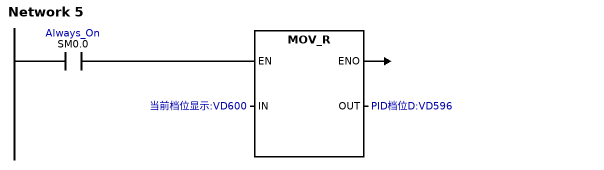
[picture p24: SBR12 networks 5-5]
Network 5
LD     Always_On:SM0.0
MOVR   当前档位显示:VD600, PID档位D:VD596
END_SUBROUTINE_BLOCK

SUBROUTINE_BLOCK PID换算档位:SBR13
TITLE=
BEGIN
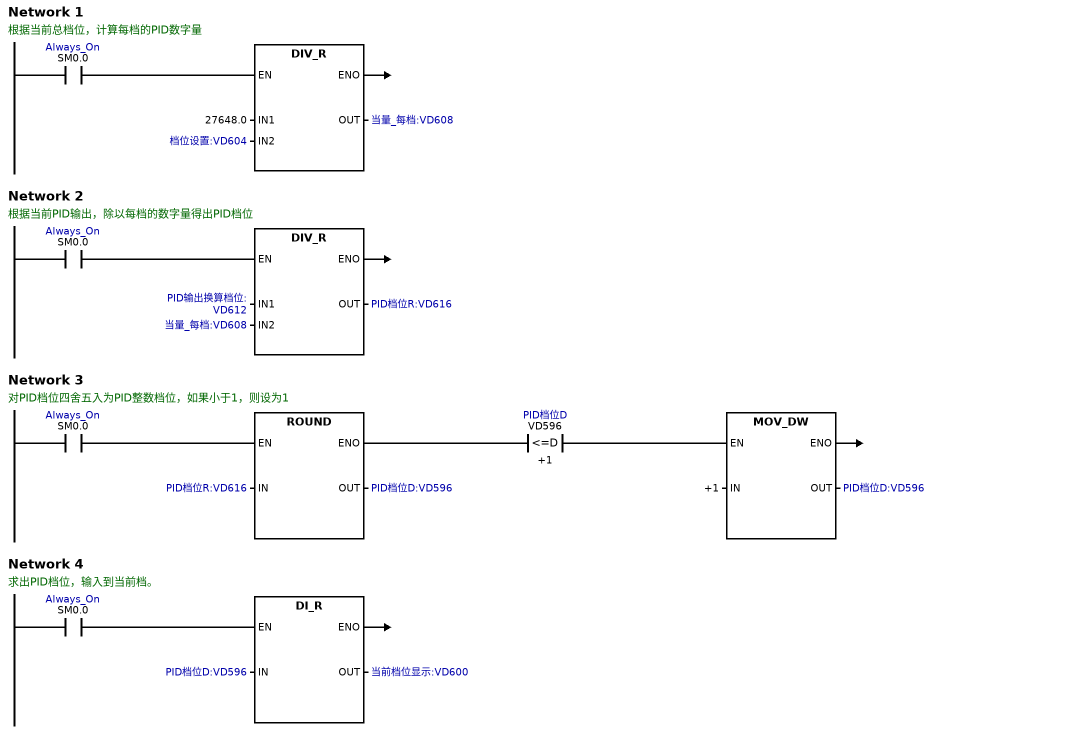
Network 1
// 根据当前总档位，计算每档的PID数字量
LD     Always_On:SM0.0
MOVR   27648.0, 当量_每档:VD608
/R     档位设置:VD604, 当量_每档:VD608
Network 2
// 根据当前PID输出，除以每档的数字量得出PID档位
LD     Always_On:SM0.0
MOVR   PID输出换算档位:VD612, PID档位R:VD616
/R     当量_每档:VD608, PID档位R:VD616
Network 3
// 对PID档位四舍五入为PID整数档位，如果小于1，则设为1
LD     Always_On:SM0.0
ROUND  PID档位R:VD616, PID档位D:VD596
AENO
AD<=   PID档位D:VD596, +1
MOVD   +1, PID档位D:VD596
Network 4
// 求出PID档位，输入到当前档。
LD     Always_On:SM0.0
DTR    PID档位D:VD596, 当前档位显示:VD600
END_SUBROUTINE_BLOCK

SUBROUTINE_BLOCK 数据初始化封装:SBR14
TITLE=
BEGIN
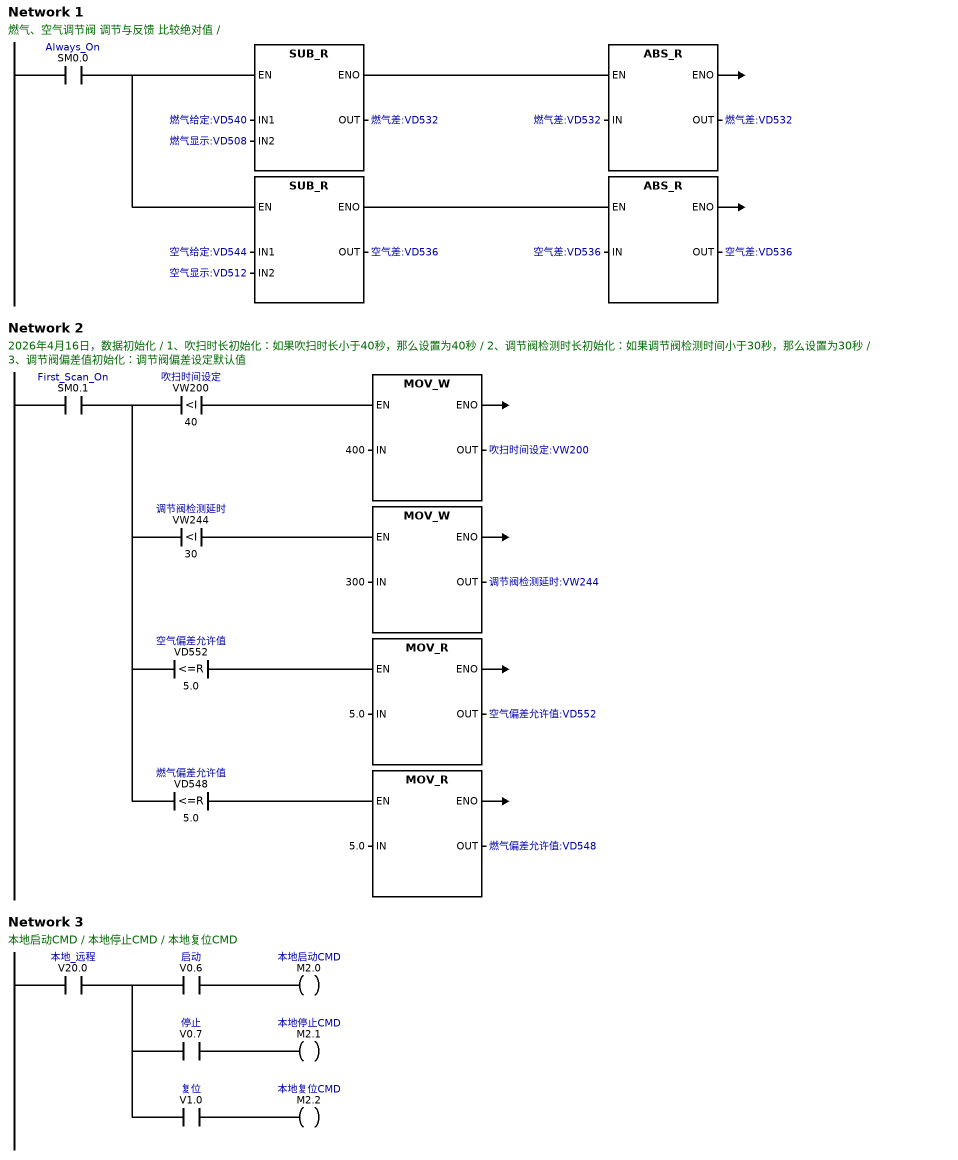
Network 1
// 燃气、空气调节阀 调节与反馈 比较绝对值
// 
LD     Always_On:SM0.0
LPS
MOVR   燃气给定:VD540, 燃气差:VD532
AENO
-R     燃气显示:VD508, 燃气差:VD532
AENO
ABSR   燃气差:VD532, 燃气差:VD532
LPP
MOVR   空气给定:VD544, 空气差:VD536
AENO
-R     空气显示:VD512, 空气差:VD536
AENO
ABSR   空气差:VD536, 空气差:VD536
Network 2
// 2026年4月16日，数据初始化
// 1、吹扫时长初始化：如果吹扫时长小于40秒，那么设置为40秒
// 2、调节阀检测时长初始化：如果调节阀检测时间小于30秒，那么设置为30秒
// 3、调节阀偏差值初始化：调节阀偏差设定默认值
LD     First_Scan_On:SM0.1
LPS
AW<    吹扫时间设定:VW200, 40
MOVW   400, 吹扫时间设定:VW200
LRD
AW<    调节阀检测延时:VW244, 30
MOVW   300, 调节阀检测延时:VW244
LRD
AR<=   空气偏差允许值:VD552, 5.0
MOVR   5.0, 空气偏差允许值:VD552
LPP
AR<=   燃气偏差允许值:VD548, 5.0
MOVR   5.0, 燃气偏差允许值:VD548
Network 3
// 本地启动CMD
// 本地停止CMD
// 本地复位CMD
LD     本地_远程:V20.0
LPS
A      启动:V0.6
=      本地启动CMD:M2.0
LRD
A      停止:V0.7
=      本地停止CMD:M2.1
LPP
A      复位:V1.0
=      本地复位CMD:M2.2
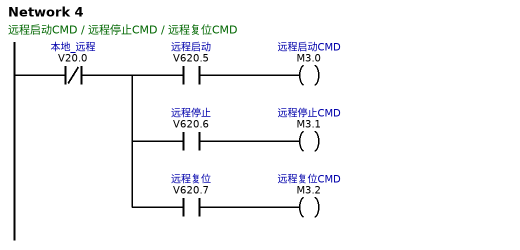
Network 4
// 远程启动CMD
// 远程停止CMD
// 远程复位CMD
LDN    本地_远程:V20.0
LPS
A      远程启动:V620.5
=      远程启动CMD:M3.0
LRD
A      远程停止:V620.6
=      远程停止CMD:M3.1
LPP
A      远程复位:V620.7
=      远程复位CMD:M3.2
END_SUBROUTINE_BLOCK

SUBROUTINE_BLOCK 报警复位停机:SBR16
TITLE=
BEGIN
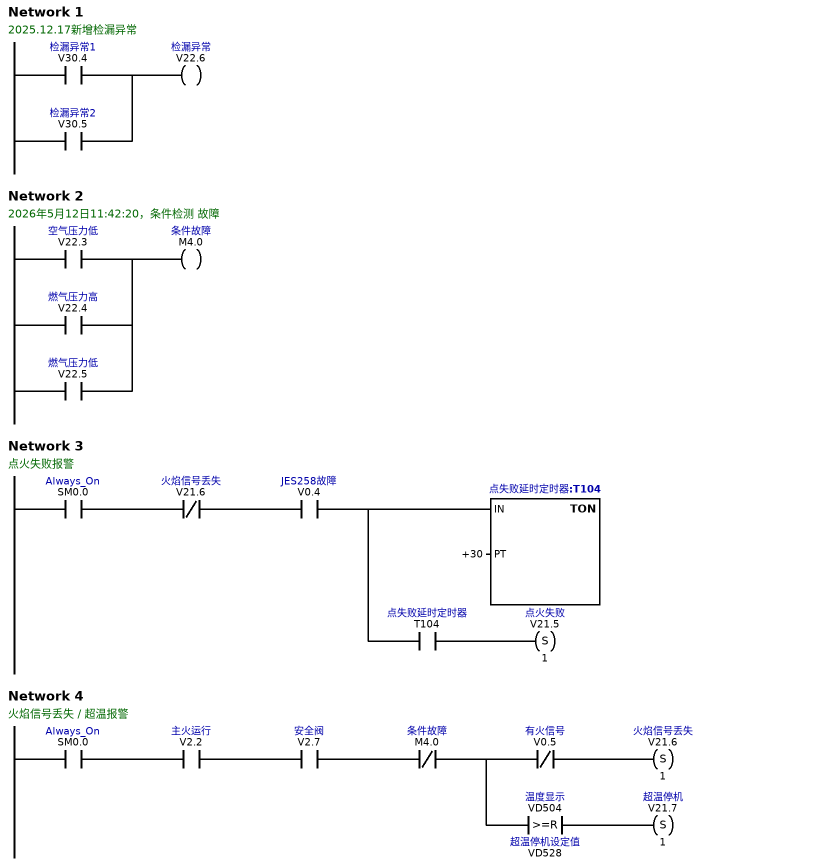
Network 1
// 2025.12.17新增检漏异常
LD     检漏异常1:V30.4
O      检漏异常2:V30.5
=      检漏异常:V22.6
Network 2
// 2026年5月12日11:42:20，条件检测 故障
LD     空气压力低:V22.3
O      燃气压力高:V22.4
O      燃气压力低:V22.5
=      条件故障:M4.0
Network 3
// 点火失败报警
LD     Always_On:SM0.0
AN     火焰信号丢失:V21.6
A      JES258故障:V0.4
TON    点失败延时定时器:T104, +30
A      点失败延时定时器:T104
S      点火失败:V21.5, 1
Network 4
// 火焰信号丢失
// 超温报警
LD     Always_On:SM0.0
A      主火运行:V2.2
A      安全阀:V2.7
AN     条件故障:M4.0
LPS
AN     有火信号:V0.5
S      火焰信号丢失:V21.6, 1
LPP
AR>=   温度显示:VD504, 超温停机设定值:VD528
S      超温停机:V21.7, 1
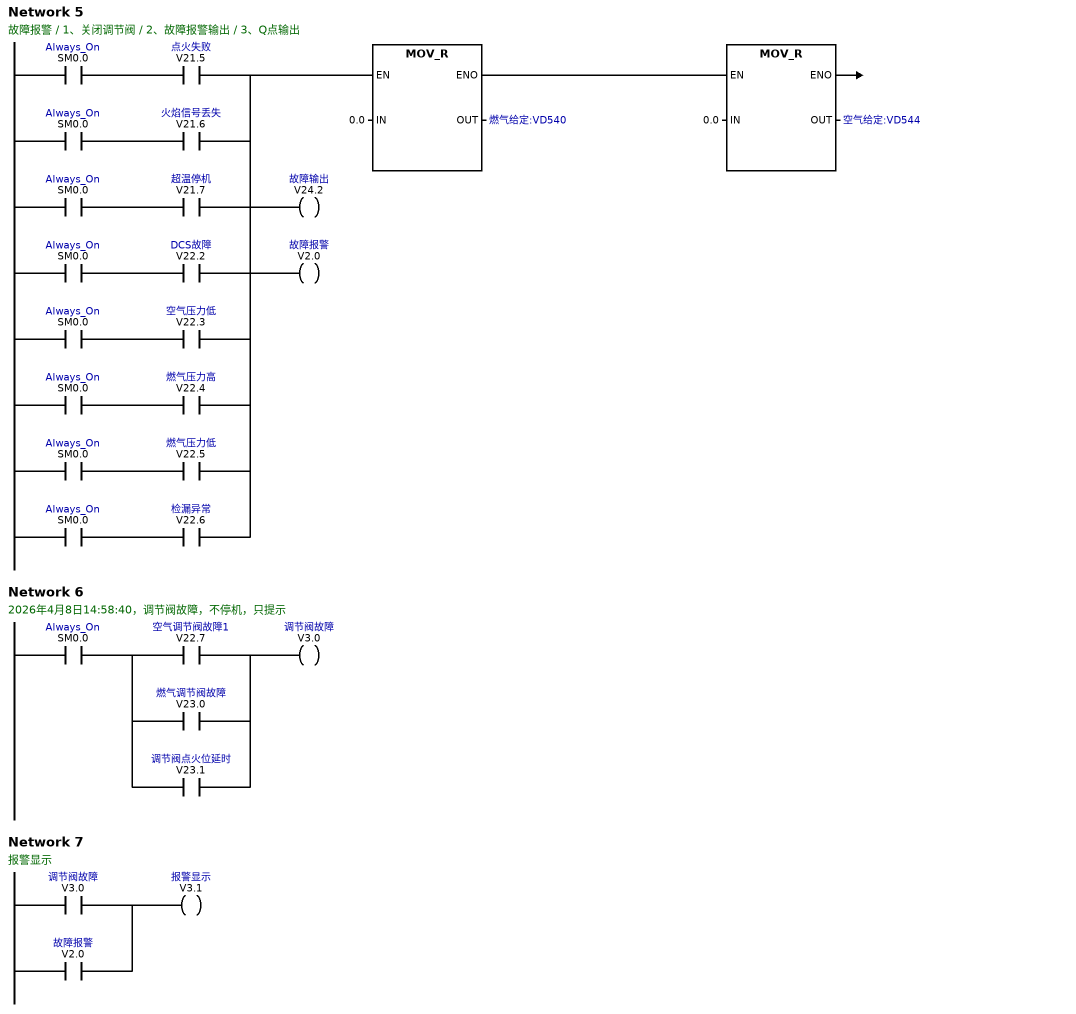
Network 5
// 故障报警
// 1、关闭调节阀
// 2、故障报警输出
// 3、Q点输出
LD     Always_On:SM0.0
A      点火失败:V21.5
LD     Always_On:SM0.0
A      火焰信号丢失:V21.6
OLD
LD     Always_On:SM0.0
A      超温停机:V21.7
OLD
LD     Always_On:SM0.0
A      DCS故障:V22.2
OLD
LD     Always_On:SM0.0
A      空气压力低:V22.3
OLD
LD     Always_On:SM0.0
A      燃气压力高:V22.4
OLD
LD     Always_On:SM0.0
A      燃气压力低:V22.5
OLD
LD     Always_On:SM0.0
A      检漏异常:V22.6
OLD
LPS
MOVR   0.0, 燃气给定:VD540
AENO
MOVR   0.0, 空气给定:VD544
LRD
=      故障输出:V24.2
LPP
=      故障报警:V2.0
Network 6
// 2026年4月8日14:58:40，调节阀故障，不停机，只提示
LD     Always_On:SM0.0
LD     空气调节阀故障1:V22.7
O      燃气调节阀故障:V23.0
O      调节阀点火位延时:V23.1
ALD
=      调节阀故障:V3.0
Network 7
// 报警显示
LD     调节阀故障:V3.0
O      故障报警:V2.0
=      报警显示:V3.1
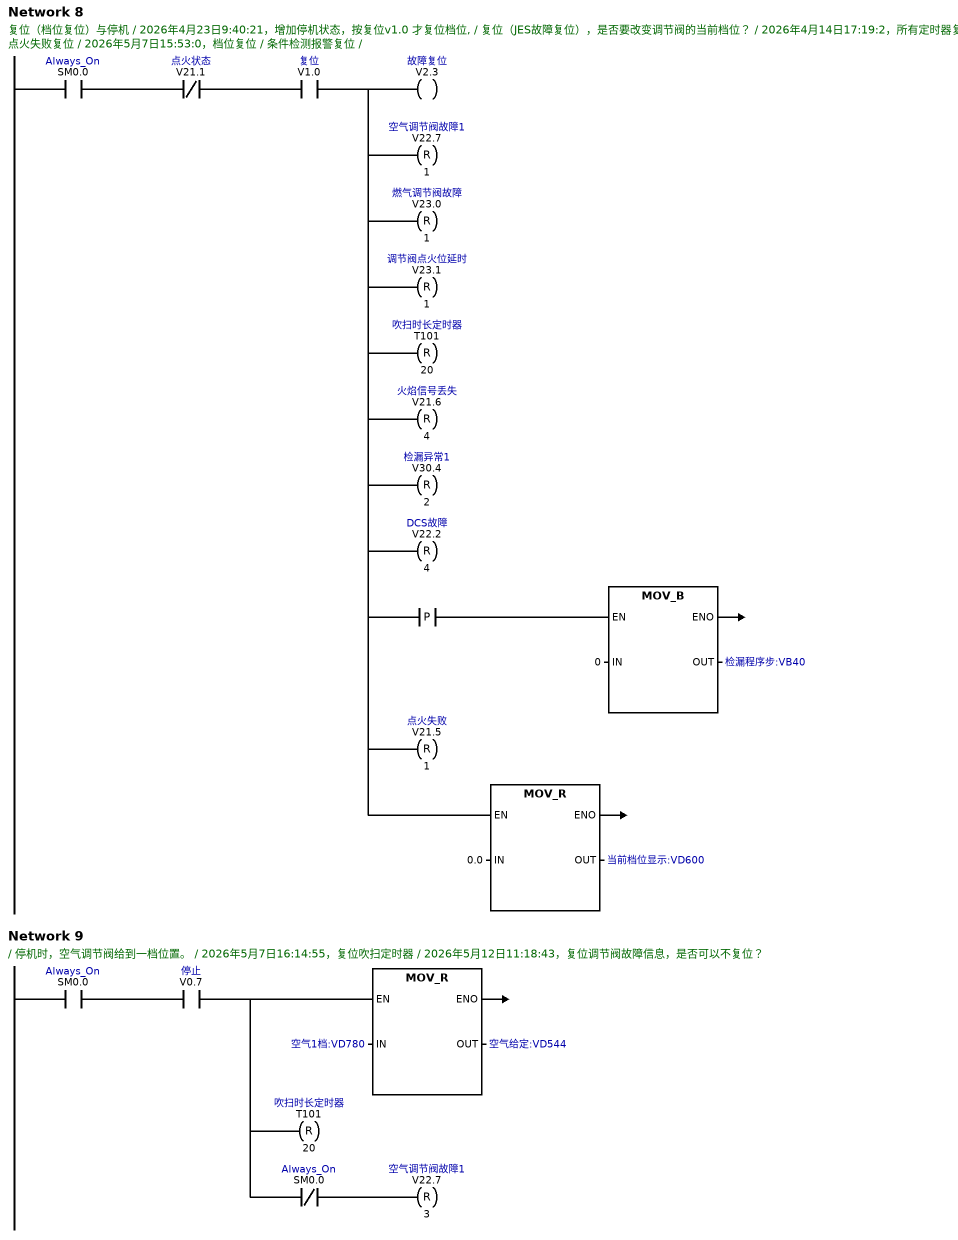
Network 8
// 复位（档位复位）与停机
// 2026年4月23日9:40:21，增加停机状态，按复位v1.0 才复位档位,
// 复位（JES故障复位），是否要改变调节阀的当前档位？
// 2026年4月14日17:19:2，所有定时器复位？
// 报警复位、检漏复位
// 点火失败复位
// 2026年5月7日15:53:0，档位复位
// 条件检测报警复位
// 
LD     Always_On:SM0.0
AN     点火状态:V21.1
A      复位:V1.0
LPS
=      故障复位:V2.3
R      空气调节阀故障1:V22.7, 1
R      燃气调节阀故障:V23.0, 1
R      调节阀点火位延时:V23.1, 1
R      吹扫时长定时器:T101, 20
R      火焰信号丢失:V21.6, 4
R      检漏异常1:V30.4, 2
R      DCS故障:V22.2, 4
EU
MOVB   0, 检漏程序步:VB40
LRD
R      点火失败:V21.5, 1
LPP
MOVR   0.0, 当前档位显示:VD600
Network 9
// 
// 停机时，空气调节阀给到一档位置。
// 2026年5月7日16:14:55，复位吹扫定时器
// 2026年5月12日11:18:43，复位调节阀故障信息，是否可以不复位？
LD     Always_On:SM0.0
A      停止:V0.7
MOVR   空气1档:VD780, 空气给定:VD544
R      吹扫时长定时器:T101, 20
AN     Always_On:SM0.0
R      空气调节阀故障1:V22.7, 3
END_SUBROUTINE_BLOCK

// SBR17: protected block, not included

// SBR18: protected block, not included

SUBROUTINE_BLOCK 通讯地址:SBR19
TITLE=子程序注释
BEGIN
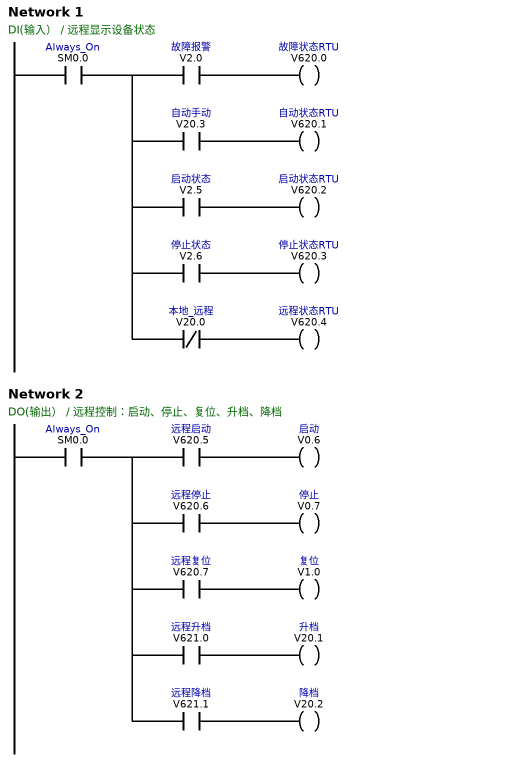
Network 1
// DI(输入）
// 远程显示设备状态
LD     Always_On:SM0.0
LPS
A      故障报警:V2.0
=      故障状态RTU:V620.0
LRD
A      自动手动:V20.3
=      自动状态RTU:V620.1
LRD
A      启动状态:V2.5
=      启动状态RTU:V620.2
LRD
A      停止状态:V2.6
=      停止状态RTU:V620.3
LPP
AN     本地_远程:V20.0
=      远程状态RTU:V620.4
Network 2
// DO(输出）
// 远程控制：启动、停止、复位、升档、降档
LD     Always_On:SM0.0
LPS
A      远程启动:V620.5
=      启动:V0.6
LRD
A      远程停止:V620.6
=      停止:V0.7
LRD
A      远程复位:V620.7
=      复位:V1.0
LRD
A      远程升档:V621.0
=      升档:V20.1
LPP
A      远程降档:V621.1
=      降档:V20.2
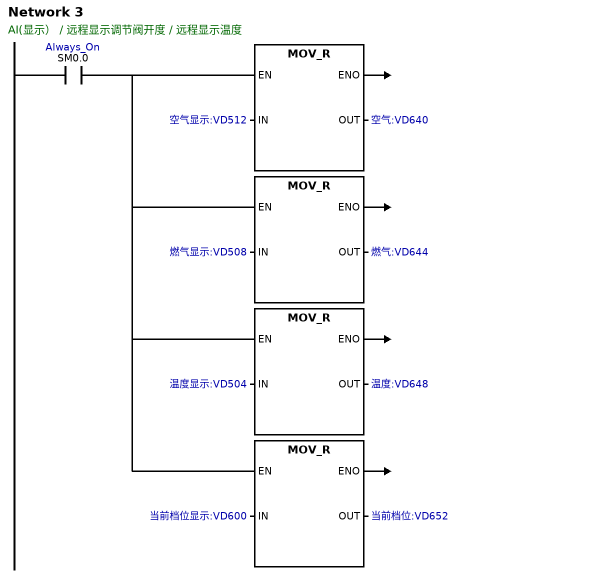
Network 3
// AI(显示）
// 远程显示调节阀开度
// 远程显示温度
LD     Always_On:SM0.0
MOVR   空气显示:VD512, 空气:VD640
MOVR   燃气显示:VD508, 燃气:VD644
MOVR   温度显示:VD504, 温度:VD648
MOVR   当前档位显示:VD600, 当前档位:VD652
END_SUBROUTINE_BLOCK

// INT0: protected block, not included

DATA_BLOCK_TAB 页面_1
BEGIN
//数据页注释
//按 F1 获取帮助和示例数据页
         阶段1温度, 0.0
         阶段2温度, 0.0
         阶段3温度, 0.0
         阶段4温度, 0.0
         阶段5温度, 0.0
         阶段6温度, 500.0
         阶段1设定, 0
         阶段2设定, 0
         阶段3设定, 0
         阶段4设定, 0
         阶段5设定, 0
         阶段6设定, 1
         温度上限设定值, 999.0
         超温停机设定值, 985.0
         PID增益_P, 17.0
         PID积分_I, 10.0
         PID微分_D, 0
         PID采样时间, 0.01
         燃气3档_1档, 15.0
         燃气4档, 20.0
         燃气5档, 25.0
         燃气6档, 30.0
         燃气7档, 35.0
         燃气8档, 40.0
         燃气9档, 45.0
         燃气10档, 50.0
         燃气11档, 55.0
         燃气12档, 60.0
         燃气13档, 65.0
         燃气14档, 70.0
         燃气15档, 75.0
         燃气16档, 80.0
         空气3档, 15.0
         空气4档, 20.0
         空气5档, 25.0
         空气6档, 30.0
         空气7档, 35.0
         空气8档, 40.0
         空气9档, 45.0
         空气10档, 50.0
         空气11档, 55.0
         空气12档, 60.0
         空气13档, 65.0
         空气14档, 70.0
         空气15档, 75.0
         空气16档, 80.0
         档位设置, 14.0
         吹扫时间设定, 9
         吹扫空气阀开度, 80.0
         空气2档, 10.0
         点火延时设定值, 9
         主火阀开启延时, 9
END_DATA_BLOCK_TAB
